Yaskawa INFORM job: R2_W63-A1(120,-90)AWOK.JBI

/JOB
//NAME R2_W63-A1(120,-90)AWOK
///FOLDERNAME AWOK
//POS
///NPOS 41,41,0,3,0,0
///TOOL 0
///POSTYPE PULSE
///PULSE
C00000=120300,89472,27287,17633,86752,-9277
C00001=132514,57588,51166,3335,64132,-22344
C00002=133277,65412,63365,3186,60620,-22157
C00003=133575,69043,68948,3135,59040,-22087
C00004=133561,69987,70620,3157,58497,-22108
C00005=133575,69043,68948,3135,59040,-22087
C00006=134027,70538,70008,2978,59140,-21910
C00007=133966,72658,72528,3013,58679,-21945
C00008=134019,71785,71849,2996,58648,-21926
C00009=134655,67856,68069,2771,58932,-21671
C00010=135315,68205,68178,2543,59022,-21413
C00011=134655,67856,68069,2771,58932,-21671
C00012=134364,64245,62527,2826,60495,-21744
C00013=133617,56437,50387,2982,63977,-21937
C00014=136550,64495,59087,-22886,74494,38256
C00015=134961,69023,67409,-22985,71469,38254
C00016=134332,71146,71156,-23055,70172,38275
C00017=134263,73668,74643,-23162,69368,38413
C00018=134332,71146,71156,-23055,70172,38275
C00019=134254,69326,70573,-23123,69618,38359
C00020=134281,69130,70915,-23170,69338,38426
C00021=134254,69561,71112,-23152,69423,38398
C00022=134112,68260,66565,-22854,71352,37954
C00023=133413,67694,65903,-22742,71267,37703
C00024=134112,68260,66565,-22854,71352,37954
C00025=134744,66324,63078,-22805,72591,37948
C00026=136340,62145,55241,-22748,75508,37978
C00027=161901,33575,28398,-1961,45759,12769
C00028=161901,33575,28398,-1961,45759,12769
C00029=157712,69504,73977,5219,46620,10491
C00030=158501,49549,56228,-16946,45407,14810
C00031=158535,50209,58031,-17189,44676,14967
C00032=162086,66974,70955,-12551,48710,25102
C00033=132594,28161,29027,3125,52864,12174
C00034=134499,29650,30500,-12644,54647,25325
C00035=137247,28590,22655,-13256,59267,25882
C00036=137247,26354,8583,-12431,66599,25041
C00037=137179,26972,-5490,-11778,74945,24094
C00038=123752,40797,12800,-2593,-17601,8904
C00039=83359,20776,-28758,17644,86757,-9277
C00040=71074,-2070,-47397,17648,86758,-9277
BC00000=310844,232565,1074715
BC00001=311018,76824,1074561
BC00002=311018,76824,1074561
BC00003=311018,76824,1074561
BC00004=311018,76824,1074561
BC00005=311018,76824,1074561
BC00006=311018,76824,1074561
BC00007=311018,76824,1074561
BC00008=311018,76824,1074561
BC00009=311018,76824,1074561
BC00010=311018,76824,1074561
BC00011=311018,76824,1074561
BC00012=311018,76824,1074561
BC00013=311018,76824,1074561
BC00014=373182,63287,1070522
BC00015=373182,63287,1070522
BC00016=373182,63287,1070522
BC00017=373182,63287,1070522
BC00018=373182,63287,1070522
BC00019=373182,63287,1070522
BC00020=373182,63287,1070522
BC00021=373182,63287,1070522
BC00022=373182,63287,1070522
BC00023=373182,63287,1070522
BC00024=373182,63287,1070522
BC00025=373182,63287,1070522
BC00026=373182,63287,1070522
BC00027=398174,59607,1065768
BC00028=398174,59607,1065768
BC00029=398174,59607,1065768
BC00030=398174,59632,1075175
BC00031=398174,59632,1075175
BC00032=398174,59607,1065768
BC00033=398174,59608,1065766
BC00034=398174,59608,1065766
BC00035=398174,59608,1065766
BC00036=398174,59608,1065766
BC00037=398088,59611,1065803
BC00038=376123,513022,1075174
BC00039=286764,353416,1074713
BC00040=278756,393608,1074712
///POSTYPE BASE
///RECTAN
///RCONF 0,0,0,0,0,0,0,0,0,0,0,0,0,0,0,0,0,0,0,0,0,0,0,0
P00006=0.222,-3.123,-1.508,0.0000,0.0000,0.0000
P00021=-0.225,-6.128,-0.405,0.0000,0.0000,0.0000
P00022=0.222,-3.123,-1.508,0.0000,0.0000,0.0000
//INST
///DATE 2023/11/16 10:55
///ATTR SC,RW
///GROUP1 RB1,BS1
NOP
'SEARCH DO POPRAWY
'SEARCH DO POPRAWY
'SEARCH DO POPRAWY
'SEARCH DO POPRAWY
'SEARCH DO POPRAWY
'pochylenie palnika do poprawy
'r2_W63-A1(120.-90)
'Path S1152
SFTOF
MOVJ C00000 BC00000 VJ=20.00
MOVJ C00001 BC00001 VJ=20.00
MOVL C00002 BC00002 V=100.0
MOVL C00003 BC00003 V=60.0
REFP 3 C00004 BC00004
CALL JOB:SEARCH-R1
SET P021 P006
SFTON P021
MOVL C00005 BC00005 V=60.0
MOVL C00006 BC00006 V=60.0
REFP 3 C00007 BC00007
CALL JOB:SEARCH-R1
SET P021 P006
SFTON P021
MOVL C00008 BC00008 V=60.0
MOVL C00009 BC00009 V=60.0
REFP 3 C00010 BC00010
CALL JOB:SEARCH-R1
SET P021 P006
SFTON P021
MOVL C00011 BC00011 V=60.0
MOVL C00012 BC00012 V=100.0
MOVL C00013 BC00013 V=100.0
'Path S1153
SFTOF
MOVJ C00014 BC00014 VJ=20.00
MOVL C00015 BC00015 V=100.0
MOVL C00016 BC00016 V=60.0
REFP 3 C00017 BC00017
CALL JOB:SEARCH-R1
SET P022 P006
SFTON P022
MOVL C00018 BC00018 V=60.0
MOVL C00019 BC00019 V=60.0
REFP 3 C00020 BC00020
CALL JOB:SEARCH-R1
SET P022 P006
SFTON P022
MOVL C00021 BC00021 V=60.0
MOVL C00022 BC00022 V=60.0
REFP 3 C00023 BC00023
CALL JOB:SEARCH-R1
SET P022 P006
SFTON P022
MOVL C00024 BC00024 V=60.0
MOVL C00025 BC00025 V=100.0
MOVL C00026 BC00026 V=100.0
'Path W1154
SFTOF
SFTON P022
MOVJ C00027 BC00027 VJ=20.00
MOVL C00028 BC00028 V=100.0
MOVL C00029 BC00029 V=100.0 PL=0
REFP 1 C00030 BC00030
REFP 2 C00031 BC00031
MACRO1 MJ#(0) ARGF9
ARCON
MOVL C00032 BC00032 V=10.8
MOVL C00033 BC00033 V=10.8
MOVL C00034 BC00034 V=10.8
ARCOF
MOVL C00035 BC00035 V=100.0
MOVL C00036 BC00036 V=100.0
SFTOF
MOVJ C00037 BC00037 VJ=20.00
MOVJ C00038 BC00038 VJ=20.00
MOVJ C00039 BC00039 VJ=20.00
MOVJ C00040 BC00040 VJ=20.00
SFTOF
END
